Staubli VAL3: GenericPage.dtx

num nCOLMAX = 39
num nCOLMIN
public num nColumn
public num nFocused
public num nListSize
num nROWMAX = 12
num nROWMIN
public num nRow
string sErrorMessage
string sErrorMsg[10]
  [0] = "An error has been detected in the Page library *\../*"
  [2] = "Variable sTxtBoxLen[*] has an illegal value"
  [3] = "Variable sTxtBoxPos[*] has an illegal value"
public string sFALSE = "FALSE"
public string sLabel = "-This is a label"
public string sLabelPos = "0;0"
public string sMenu = "F1 F2 ; F4 F5 F6 ; F8"
public string sTRUE = "TRUE"
public string sTitle = "custom EntryBox"
public string sTxtBoxAuthord[3] = "0123456789.-"
public string sTxtBoxCaption[3]
  [0] = "Numeric :"
  [1] = "Boolean :"
  [2] = "List    :"
public string sTxtBoxLen[3]
  [0] = "7"
  [1] = "7"
  [2] = "7"
public string sTxtBoxPos[3]
  [0] = "0;1"
  [1] = "0;2"
  [2] = "0;3"
public string sTxtBoxRange[3] = "-100;100"
public string sTxtBoxType[3]
  [0] = "N"
  [1] = "B"
  [2] = "L6;17;8;5"
public string sTxtBoxVal[3]
  [0] = "421"
  [2] = "0"
public string sListItem0
